INTERFACE I_PUMP EXTENDS I_ENGINE

END_INTERFACE

(* stored: Version 1.1.0.1, ProductVersion 3.1.4024.12
   Itf I_PUMP: Id {693c6b06-84c8-4645-a803-24b388095653} *)
